// Mitsubishi GX Works2 project: plc1008_factory_countV2   PLC: Q02/Q02H

PROGRAM MAIN
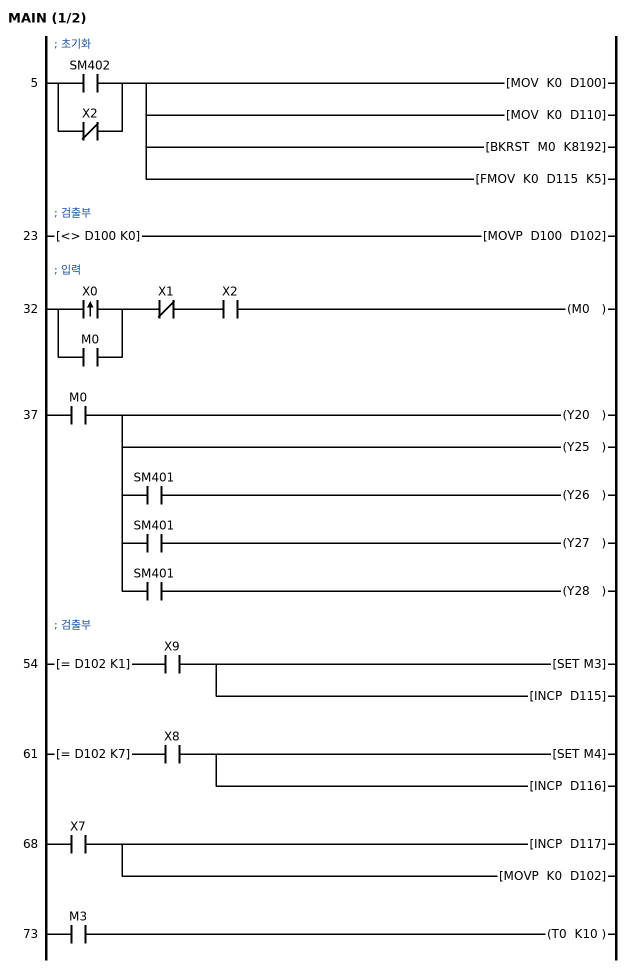
; 초기화
5     LD      SM402
      ORI     X2
      MOV     K0 D100
      MOV     K0 D110
      BKRST   M0 K8192
      FMOV    K0 D115 K5
; 검출부
23    LD<>    D100 K0
      MOVP    D100 D102
; 입력
32    LDP     X0
      OR      M0
      ANI     X1
      AND     X2
      OUT     M0
37    LD      M0
      OUT     Y20
      OUT     Y25
      MPS
      AND     SM401
      OUT     Y26
      MRD
      AND     SM401
      OUT     Y27
      MPP
      AND     SM401
      OUT     Y28
; 검출부
54    LD=     D102 K1
      AND     X9
      SET     M3
      INCP    D115
61    LD=     D102 K7
      AND     X8
      SET     M4
      INCP    D116
68    LD      X7
      INCP    D117
      MOVP    K0 D102
73    LD      M3
      OUT     T0 K10
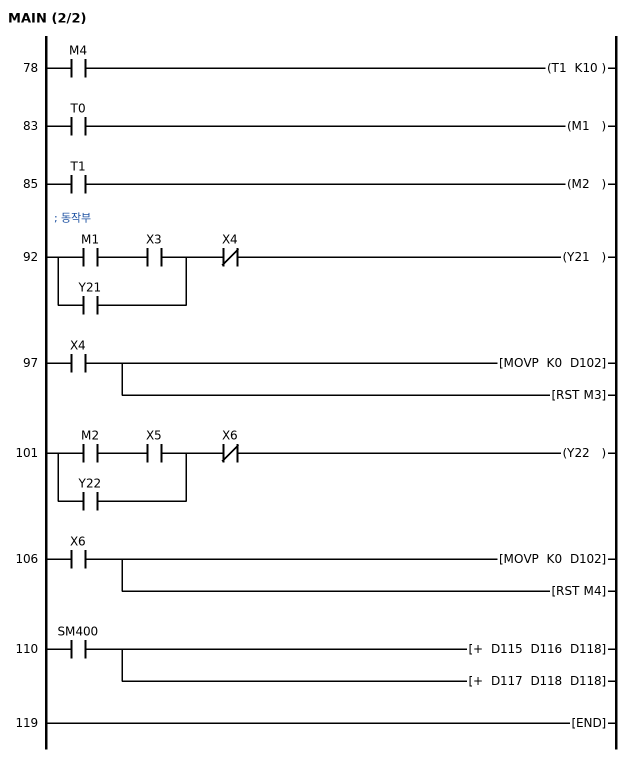
78    LD      M4
      OUT     T1 K10
83    LD      T0
      OUT     M1
85    LD      T1
      OUT     M2
; 동작부
92    LD      M1
      AND     X3
      OR      Y21
      ANI     X4
      OUT     Y21
97    LD      X4
      MOVP    K0 D102
      RST     M3
101   LD      M2
      AND     X5
      OR      Y22
      ANI     X6
      OUT     Y22
106   LD      X6
      MOVP    K0 D102
      RST     M4
110   LD      SM400
      +       D115 D116 D118
      +       D117 D118 D118
119   END
END_PROGRAM
